// Mitsubishi GX Works2 project: ｃarlo   PLC: Q06H

PROGRAM MAIN
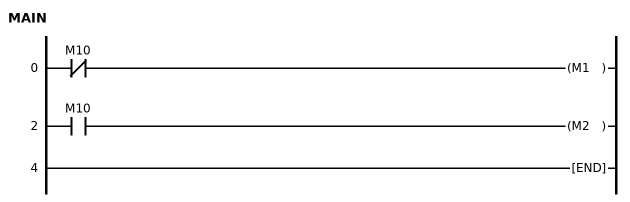
0     LDI     M10
      OUT     M1
2     LD      M10
      OUT     M2
4     END
END_PROGRAM
